Fanuc KAREL source: kx00019.compact.KL

PROGRAM KX00019
%STACKSIZE=65535
%PRIORITY=65535
%NOLOCKGROUP
VAR
I : INTEGER
J : INTEGER
B : BOOLEAN
F : FILE
S : STRING[80]
P : XYZWPR
SH : ARRAY[4] OF SHORT
BEGIN
SH[1]=123
I=SH[1]
END KX00019
